FUNCTION_BLOCK PUBLIC TmsSwitchStation EXTENDS Process
VAR_INPUT
	TmsSwitch : ITF_TmsSwitch;
END_VAR
VAR_OUTPUT
END_VAR
VAR
	movers : ARRAY[1..3] OF ITmsMover;
	StationLocation : INT := 1; //1 = low, 2 = high
END_VAR

//Station for tms handling
//these are implemented at each entry to the switch

//Do i have mover?
////Do i have switch?
//////If yes pass mover to switch
//////If mover on switch send switch
//////once station done bring rear mover forward
////Else 
//////Wait for switch
//Else
////Wait for movers

METHOD PUBLIC MoverArriving : BOOL
VAR_INPUT
	mover : IMover;
END_VAR
VAR
	iTmsMover : ITmsMover;
END_VAR
IF StationMovers <= 2 THEN
	StationMovers := StationMovers + 1;
	IF __QUERYINTERFACE(mover,iTmsMover) THEN
		movers[StationMovers] := iTmsMover;
	END_IF
END_IF
END_METHOD

METHOD PUBLIC MoverAway : BOOL
VAR_INPUT
END_VAR
IF StationMovers = 1 THEN
	StationMovers := StationMovers - 1;
	movers[1] := 0;
	movers[2] := 0;
	movers[3] := 0;
ELSIF StationMovers = 2 THEN
	StationMovers := StationMovers - 1;
	movers[1] := movers[2];
	movers[2] := 0;
	movers[3] := 0;
ELSIF StationMovers = 3 THEN
	StationMovers := StationMovers - 1;
	movers[1] := movers[2];
	movers[2] := movers[3];
	movers[3] := 0;
END_IF
END_METHOD

METHOD PUBLIC SwitchMoveComplete : BOOL
VAR_INPUT
END_VAR
_Complete := SwitchMoveComplete := true;
END_METHOD

END_FUNCTION_BLOCK

(* stored: Version 1.1.0.1, ProductVersion 3.1.4024.11
   POU TmsSwitchStation: Id {27fb18f6-f27b-4462-bf40-a5ac4ef58917}, SpecialFunc None
   Method MoverArriving: Id {9da69018-e0b3-43b6-8b40-80f26b1bd5d9}
   Method MoverAway: Id {5d30fab5-165d-4159-bdc5-36df29db049b}
   Method SwitchMoveComplete: Id {b6e4018d-1b11-4436-abf3-c2d1900106a2} *)
